// SIMATIC STEP 7 (V5.x) project P_P_Pr01
// program: S7 Program(1)

SYMBOL_TABLE
"PART_AV"	I 0.0	BOOL
"Sli_Back"	I 0.1	BOOL
"Sli_Frnt"	I 0.2	BOOL
"Sli_Up"	I 0.3	BOOL
"Sen_Vac"	I 0.4	BOOL
"Wp_Pro"	I 0.5	BOOL
"Wp_End"	I 0.6	BOOL
"START"	I 1.0	BOOL
"STOP"	I 1.1	BOOL
"AUTOMAN"	I 1.2	BOOL
"RESET"	I 1.3	BOOL
"Conveyor"	Q 0.0	BOOL
"SliBack"	Q 0.1	BOOL
"SliFrnt"	Q 0.2	BOOL
"SliDown"	Q 0.3	BOOL
"Vacuum"	Q 0.4	BOOL
"Separator"	Q 0.5	BOOL
"L_Q1"	Q 1.2	BOOL
"L_Q2"	Q 1.3	BOOL
END_SYMBOL_TABLE

FUNCTION FC 1 : VOID
VERSION : 0.1
BEGIN
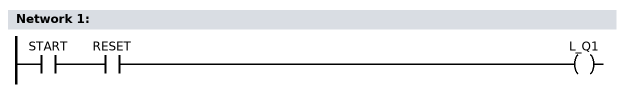
NETWORK
TITLE =
      A     "START";
      A     "RESET";
      =     "L_Q1";
END_FUNCTION

FUNCTION FC 2 : VOID
VERSION : 0.1
BEGIN
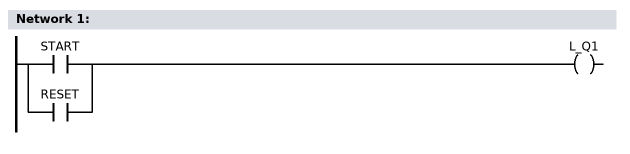
NETWORK
TITLE =
      O     "START";
      O     "RESET";
      =     "L_Q1";
END_FUNCTION

FUNCTION FC 3 : VOID
VERSION : 0.1
BEGIN
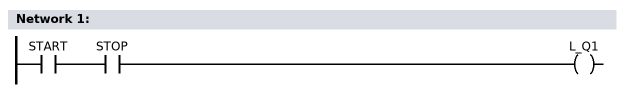
NETWORK
TITLE =
      A     "START";
      A     "STOP";
      =     "L_Q1";
END_FUNCTION

FUNCTION FC 4 : VOID
VERSION : 0.1
BEGIN
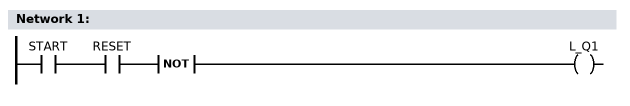
NETWORK
TITLE =
      A     "START";
      A     "RESET";
      NOT;
      =     "L_Q1";
END_FUNCTION

FUNCTION FC 5 : VOID
VERSION : 0.1
BEGIN
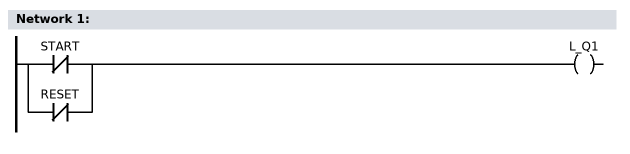
NETWORK
TITLE =
      ON    "START";
      ON    "RESET";
      =     "L_Q1";
NETWORK
TITLE =
END_FUNCTION

FUNCTION FC 6 : VOID
VERSION : 0.1
BEGIN
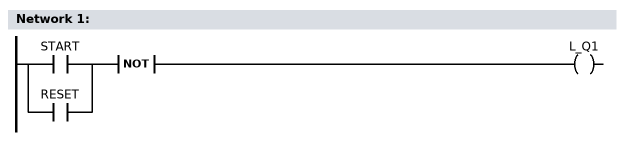
NETWORK
TITLE =
      A(;
      O     "START";
      O     "RESET";
      );
      NOT;
      =     "L_Q1";
END_FUNCTION

FUNCTION FC 7 : VOID
VERSION : 0.1
BEGIN
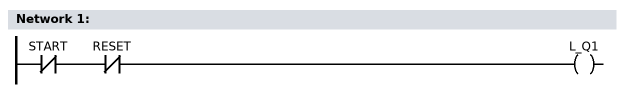
NETWORK
TITLE =
      AN    "START";
      AN    "RESET";
      =     "L_Q1";
END_FUNCTION

FUNCTION FC 8 : VOID
VERSION : 0.1
BEGIN
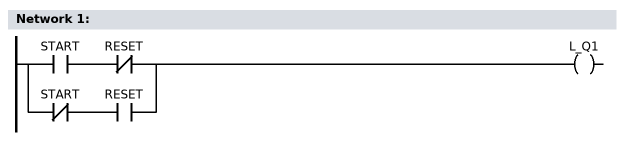
NETWORK
TITLE =
      A     "START";
      AN    "RESET";
      O;
      AN    "START";
      A     "RESET";
      =     "L_Q1";
END_FUNCTION

FUNCTION FC 9 : VOID
VERSION : 0.1
BEGIN
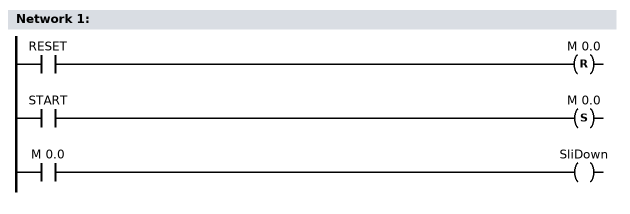
NETWORK
TITLE =
      A     "RESET";
      R     M 0.0;
      A     "START";
      S     M 0.0;
      A     M 0.0;
      =     "SliDown";
END_FUNCTION

FUNCTION FC 10 : VOID
VERSION : 0.1
BEGIN
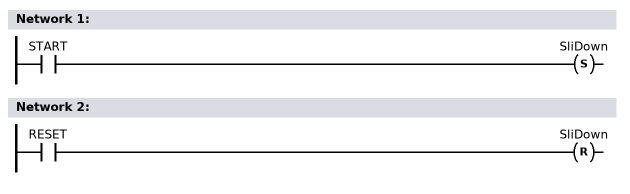
NETWORK
TITLE =
      A     "START";
      S     "SliDown";
NETWORK
TITLE =
      A     "RESET";
      R     "SliDown";
END_FUNCTION

FUNCTION FC 11 : VOID
VERSION : 0.1
BEGIN
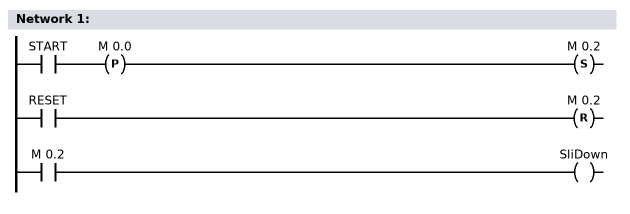
NETWORK
TITLE =
      A     "START";
      FP    M 0.0;
      S     M 0.2;
      A     "RESET";
      R     M 0.2;
      A     M 0.2;
      =     "SliDown";
END_FUNCTION

FUNCTION FC 12 : VOID
VERSION : 0.1
BEGIN
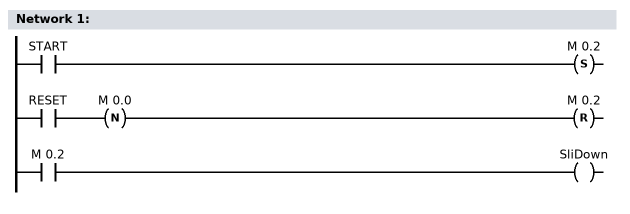
NETWORK
TITLE =
      A     "START";
      S     M 0.2;
      A     "RESET";
      FN    M 0.0;
      R     M 0.2;
      A     M 0.2;
      =     "SliDown";
END_FUNCTION

FUNCTION FC 13 : VOID
VERSION : 0.1
BEGIN
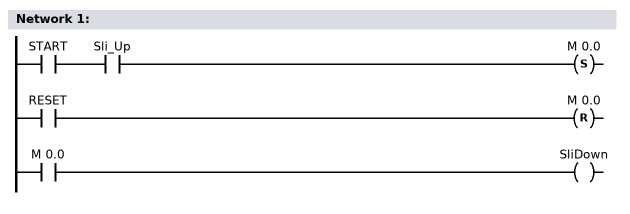
NETWORK
TITLE =
      A     "START";
      A     "Sli_Up";
      S     M 0.0;
      A     "RESET";
      R     M 0.0;
      A     M 0.0;
      =     "SliDown";
END_FUNCTION

FUNCTION FC 14 : VOID
VERSION : 0.1
BEGIN
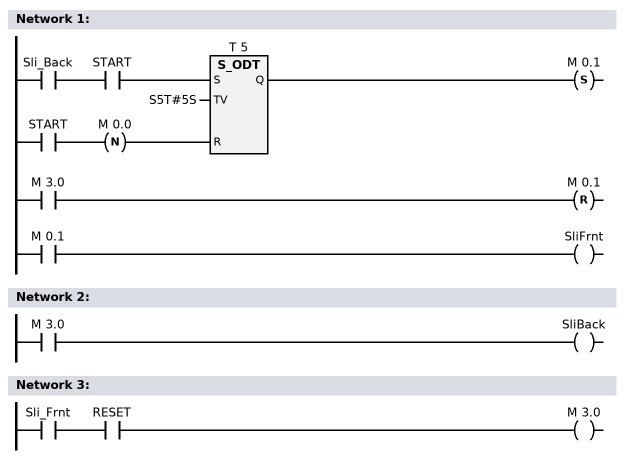
NETWORK
TITLE =
      A(;
      A     "Sli_Back";
      A     "START";
      L     S5T#5S;
      SD    T 5;
      A     "START";
      FN    M 0.0;
      R     T 5;
      NOP   0;
      NOP   0;
      A     T 5;
      );
      S     M 0.1;
      A     M 3.0;
      R     M 0.1;
      A     M 0.1;
      =     "SliFrnt";
NETWORK
TITLE =
      A     M 3.0;
      =     "SliBack";
NETWORK
TITLE =
      A     "Sli_Frnt";
      A     "RESET";
      =     M 3.0;
END_FUNCTION

FUNCTION FC 15 : VOID
VERSION : 0.1
BEGIN
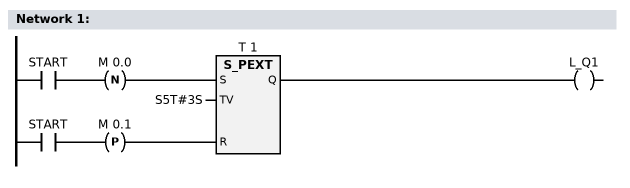
NETWORK
TITLE =
      A     "START";
      FN    M 0.0;
      L     S5T#3S;
      SE    T 1;
      A     "START";
      FP    M 0.1;
      R     T 1;
      NOP   0;
      NOP   0;
      A     T 1;
      =     "L_Q1";
END_FUNCTION

FUNCTION FC 16 : VOID
VERSION : 0.1
BEGIN
NETWORK
TITLE =
      A(;
      A     "START";
      CD    C 1;
      BLD   101;
      A     "RESET";
      L     C#5;
      S     C 1;
      AN    "STOP";
      R     C 1;
      NOP   0;
      NOP   0;
      A     C 1;
      );
      NOT;
      =     "L_Q1";
NETWORK
TITLE =
END_FUNCTION

FUNCTION FC 17 : VOID
VERSION : 0.1
BEGIN
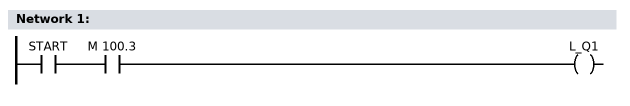
NETWORK
TITLE =
      A     "START";
      A     M 100.3;
      =     "L_Q1";
END_FUNCTION

FUNCTION FC 18 : VOID
VERSION : 0.1
BEGIN
NETWORK
TITLE =
      A(;
      A     "START";
      A     "Sli_Back";
      CU    C 1;
      BLD   101;
      A     "RESET";
      L     C#1;
      S     C 1;
      NOP   0;
      NOP   0;
      NOP   0;
      A     C 1;
      );
      S     M 0.0;
      A     M 1.0;
      R     M 0.0;
      A     M 0.0;
      =     "SliFrnt";
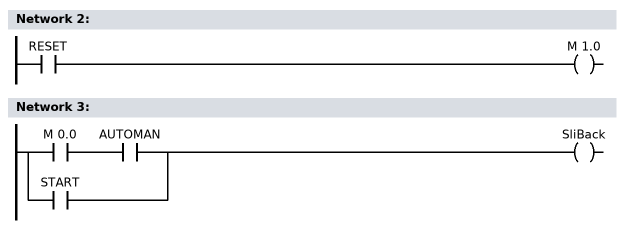
NETWORK
TITLE =
      A     "RESET";
      =     M 1.0;
NETWORK
TITLE =
      A     M 0.0;
      A     "AUTOMAN";
      O     "START";
      =     "SliBack";
END_FUNCTION

ORGANIZATION_BLOCK OB 1
TITLE = "Main Program Sweep (Cycle)"
VERSION : 0.1
VAR_TEMP
  OB1_EV_CLASS : BYTE ;	//Bits 0-3 = 1 (Coming event), Bits 4-7 = 1 (Event class 1)
  OB1_SCAN_1 : BYTE ;	//1 (Cold restart scan 1 of OB 1), 3 (Scan 2-n of OB 1)
  OB1_PRIORITY : BYTE ;	//Priority of OB Execution
  OB1_OB_NUMBR : BYTE ;	//1 (Organization block 1, OB1)
  OB1_RESERVED_1 : BYTE ;	//Reserved for system
  OB1_RESERVED_2 : BYTE ;	//Reserved for system
  OB1_PREV_CYCLE : INT ;	//Cycle time of previous OB1 scan (milliseconds)
  OB1_MIN_CYCLE : INT ;	//Minimum cycle time of OB1 (milliseconds)
  OB1_MAX_CYCLE : INT ;	//Maximum cycle time of OB1 (milliseconds)
  OB1_DATE_TIME : DATE_AND_TIME ;	//Date and time OB1 started
END_VAR
BEGIN
NETWORK
TITLE =
      UC    FC 18;
END_ORGANIZATION_BLOCK
